FUNCTION_BLOCK SignalProvider
VAR_INPUT
END_VAR
VAR_OUTPUT
END_VAR
VAR
	// hashtable of signals
	// register method creates new signal and saves pointer to hashtable
	// register and retrieve signal by its pointer
	
	mappings		: ARRAY[0..10] OF SignalMapping;
	count			: INT;
	lastMapping		: REFERENCE TO SignalMapping;
END_VAR


METHOD Call : BOOL
VAR_INPUT
END_VAR
VAR
	i		: INT;
END_VAR

FOR i := 0 TO count - 1 DO
	
	mappings[i].signal^.Call();
END_FOR
END_METHOD


METHOD FB_exit : BOOL
VAR_INPUT
	bInCopyCode : BOOL; // if TRUE, the exit method is called for exiting an instance that is copied afterwards (online change).
END_VAR
VAR
	i	: INT;
END_VAR

FOR i := 0 TO count DO
	
	__DELETE(mappings[i].signal);
END_FOR
END_METHOD


METHOD Find : INT
VAR_INPUT
	symbol	: REFERENCE TO BOOL;
END_VAR
VAR
	address	: POINTER TO SignalBundle;
	i		: INT;
END_VAR

Find := -1;

address := ADR(symbol);

FOR i := 0 TO count - 1 DO
	IF mappings[i].symbol = address THEN
		
		Find := i;

		RETURN;
	END_IF
END_FOR
END_METHOD


METHOD Get : REFERENCE TO SignalBundle
VAR_INPUT
	symbol	: REFERENCE TO BOOL;
END_VAR
VAR
	found	: INT;
END_VAR

found := Find(symbol);

IF (__ISVALIDREF(lastMapping) AND_THEN ADR(symbol) = lastMapping.symbol) THEN
	
	Get REF= lastMapping.signal^;
ELSIF (found = -1) THEN
	
	Get REF= Register(symbol, '', FALSE);
ELSE
	
	Get REF= mappings[found].signal^;
	lastMapping REF= mappings[found];
END_IF
END_METHOD


METHOD Register : REFERENCE TO SignalBundle
VAR_INPUT
	symbol	 		: REFERENCE TO BOOL;
	create			: STRING;
	inverted		: BOOL;
END_VAR

mappings[count].symbol := ADR(symbol); // Use the fact, that address of reference is address of the referenced variable
mappings[count].signal := __NEW(SignalBundle(symbol := symbol, createAtStart := create, invertedLogic := inverted));

Register REF= mappings[count].signal^;

lastMapping REF= mappings[count];

count := count + 1;
END_METHOD

END_FUNCTION_BLOCK

(* stored: Version 1.1.0.1, ProductVersion 3.1.4024.11
   POU SignalProvider: Id {c34772f0-d050-443b-9d67-92f94521a1c7}, SpecialFunc None
   Method Call: Id {b316e55e-ac32-442d-b859-2429c6670890}
   Method FB_exit: Id {d7a180b5-aa1e-41c1-9eeb-00b4474e8d2f}
   Method Find: Id {aaa598f3-afa9-441a-ad6a-c6a75a0c1bf7}
   Method Get: Id {a580a647-5d54-42a7-95e3-e95bacb20b7e}
   Method Register: Id {de0d5821-fc53-4549-9de2-506e7021a55e} *)
